PROGRAM eStopPLC
VAR
	xSwitchSF14 AT %I* : BOOL;
	xSwitchSF15 AT %I* : BOOL;
	
	xRun 	AT %Q* : BOOL; 
	xErrAck AT %Q* : BOOL; 
END_VAR

xRun:= xSwitchSF14;
xErrAck := xSwitchSF15;

END_PROGRAM

(* stored: Version 1.1.0.1
   POU eStopPLC: Id {63542574-60fc-48cb-95d5-6b9ffb37bcbc}, SpecialFunc None *)
